TYPE csp_transfer_upstacker_carton_backstop :
STRUCT
	status: 					csp_transfer_upstacker_carton_backstop_status;	
	change_cam_phase:			LREAL;	
END_STRUCT
END_TYPE

(* stored: Version 1.1.0.1, ProductVersion 3.1.4022.12
   DUT csp_transfer_upstacker_carton_backstop: Id {482e2b25-e045-4d63-addc-1e7bb3e99155} *)
